(* CODESYS project master.project

Project tree, tasks and I/O mapping:
  Device : CODESYS Control for Raspberry Pi, 3S - Smart Software Solutions GmbH, version 3.5.8.10
    application Application
      libraries: Standard, * (System)
      task MainTask (cyclic, interval t#20ms, priority 1) calls PLC_PRG
      task VISU_TASK (cyclic, interval 100 ms, priority 31) calls VisuElems.Visu_Prg
      program PLC_PRG [ST]
      visualisation MainPage
    SoftMotion General Axis Pool
    GPIOs_A_B : GPIOs A/B, 3S - Smart Software Solutions GmbH, version 1.1.1.10
        unmapped channels: digital inputs (GPIO0..GPIO31), digital outputs (GPIO0..GPIO31)
    I²C
    SPI
    Onewire
    Camera device
      <Vacío>
    ModbusConfig : Ethernet, 3S - Smart Software Solutions GmbH, version 3.5.8.20
        settings: IPAddress = [192,168,1,66]; SubnetMask = [255,255,255,0]; GatewayAddress = [192,168,1,254]; MACAddress = [16#B8,16#27,16#EB,16#59,16#CC,16#13]; NetworkInterfaceName = 'eth0'; NetworkInterfaceName = "eth0"; SaveCommunicationSettings = FALSE
      Modbus_TCP_Master : Modbus TCP Master, 3S - Smart Software Solutions GmbH, version 3.5.8.10
          settings: AutoReconnect = TRUE
        Arduino_PLC1 : Modbus TCP Slave, 3S - Smart Software Solutions GmbH, version 3.5.7.0
            settings: Unit-ID = 1; IPAddress = [192, 168, 1, 110]; WriteCoils.Function Code = 15; WriteCoils.Read Offset = 0; WriteCoils.Read Length = 0; WriteCoils.Write Offset = 16#0000; WriteCoils.Write Length = 8; WriteCoils.Cycle Time = 1000
            unmapped channels: WriteCoils
        Arduino_PLC2 : Modbus TCP Slave, 3S - Smart Software Solutions GmbH, version 3.5.7.0
            settings: Unit-ID = 2; IPAddress = [192, 168, 1, 120]; Channel 0.Function Code = 3; Channel 0.Read Offset = 16#0000; Channel 0.Read Length = 8; Channel 0.Write Offset = 0; Channel 0.Write Length = 0; Channel 0.Cycle Time = 1000; Channel 1.Function Code = 15; Channel 1.Read Offset = 0; Channel 1.Read Length = 0; Channel 1.Write Offset = 16#0000; Channel 1.Write Length = 8; Channel 1.Cycle Time = 1000
            unmapped channels: Channel 0, Channel 1
  libraries: VisuSymbols, 3.5.8.0 (System)
  text list GlobalTextList
*)

// Device/Application/PLC_PRG
// National Autonomous University of Mexico 
// Paulo Contreras Flores
// paulo.contreras.flores@gmail.com

PROGRAM PLC_PRG
VAR
	Lamp1: BOOL; // Arduino Uno Lamp 1
	Lamp2: BOOL;  // Arduino Uno Lamp 2
	Lamp3: BOOL;  //Arduino Uno Lamp 3	
	Lamp4: BOOL; // Arduino Uno Lamp 4
	Lamp5: BOOL;  // Arduino Uno Lamp 5
	Lamp6: BOOL;  //Arduino Uno Lamp 6	
	
	Lamp10: BOOL;  //Arduino Uno Lamp 10
	Lamp20: BOOL;  //Arduino Uno Lamp 20
	Lamp30: BOOL;  //Arduino Uno Lamp 30
	
	
	Count: INT;
	varLDR: WORD;
END_VAR

// Arduino Uno

Count:=Count+1;
Lamp1:=Count<2100 OR (Count>4000 AND Count<4100);					    // red
Lamp3:=Count>2100 AND Count<3500;		// green
Lamp2:=Count>3500 AND Count<4000;		// yellow

Lamp6:=Count<1500;					// green
Lamp5:=Count>1500 AND Count<2000;		// yellow
Lamp4:=Count>2000 AND Count<4100;		// red

IF Count >4100 THEN
	Count:=0;
END_IF

 varLDR:=%IW0; (* photoresistor reading value *)

 Lamp10:=varLDR>256;
 Lamp20:=varLDR>=512;
 Lamp30:=varLDR>=768;


// Output Mapping
%QX0.0:=Lamp1;
%QX0.1:=Lamp2;
%QX0.2:=Lamp3;
%QX0.3:=Lamp4;
%QX0.4:=Lamp5;
%QX0.5:=Lamp6;

%QX1.0:=Lamp10;
%QX1.1:=Lamp20;
%QX1.2:=Lamp30;

END_PROGRAM

// Device/Application/MainPage
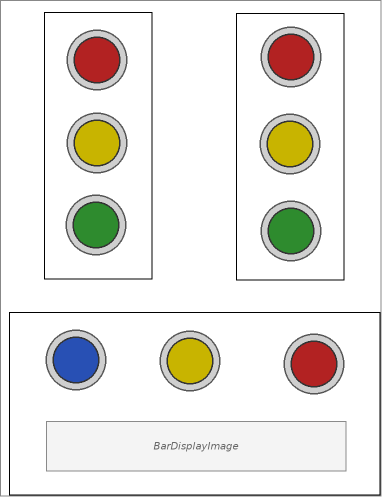
VISUALIZATION MainPage  // 382x497
    Rectangle (236,13 108x267)
    Rectangle (9,312 371x183)
    Lamp1 (41,325 70x70), variable: PLC_PRG.Lamp10, style: Lamp-Lamp1-Blue
    Lamp1 (155,326 70x70), variable: PLC_PRG.Lamp20, style: Lamp-Lamp1-Yellow
    Lamp1 (279,329 70x70), variable: PLC_PRG.Lamp30, style: Lamp-Lamp1-Red
    Rectangle (44,12 108x267)
    Lamp1 (62,108 70x70), variable: PLC_PRG.Lamp2, style: Lamp-Lamp1-Yellow
    Lamp1 (255,109 70x70), variable: PLC_PRG.Lamp5, style: Lamp-Lamp1-Yellow
    Lamp1 (62,25 70x70), variable: PLC_PRG.Lamp1, style: Lamp-Lamp1-Red
    Lamp1 (256,22 70x70), variable: PLC_PRG.Lamp4, style: Lamp-Lamp1-Red
    Lamp1 (61,190 70x70), variable: PLC_PRG.Lamp3, style: Lamp-Lamp1-Green
    Lamp1 (256,196 70x70), variable: PLC_PRG.Lamp6, style: Lamp-Lamp1-Green
    BarDisplayImage (46,421 300x50), value: PLC_PRG.varLDR, style: BarDisplayImage-Gray, scale format: %.1f, scale 0..1000
END_VISUALIZATION
